{attribute 'linkalways'} 
{attribute 'no_explicit_call' := 'This FB is a CLASS and must be accessed using methods or properties'}
{attribute 'enable_dynamic_creation'}
FUNCTION_BLOCK FINAL XOR_BYTE EXTENDS Node
VAR
	in1 : _BYTE(0);
	in2 : _BYTE(0);
	out : _BYTE(0);
END_VAR

METHOD PUBLIC Clone : I_Node
VAR
	pNode : POINTER TO XOR_BYTE;
END_VAR
pNode := __NEW(XOR_BYTE);
Clone := pNode^;
END_METHOD

METHOD FB_init : BOOL
VAR_INPUT
	bInitRetains : BOOL; // if TRUE, the retain variables are initialized (warm start / cold start)
	bInCopyCode : BOOL;  // if TRUE, the instance afterwards gets moved into the copy code (online change)
END_VAR
AddInput('in1',THIS^.in1);
AddInput('in2',THIS^.in2);
AddOutput('out', THIS^.out);
END_METHOD

METHOD PROTECTED OnExecute
VAR
END_VAR
out.Value := in1.Value XOR in2.Value;
END_METHOD

END_FUNCTION_BLOCK

(* stored: Version 1.1.0.1, ProductVersion 3.1.4024.15
   POU XOR_BYTE: Id {45796d8b-2e7a-4d20-ac19-69967073d21b}, SpecialFunc None
   Folder Constructor: Id {856a0c9a-8278-4c99-951a-6edf8ae1711c}
   Method Clone: Id {8dffed33-be2a-44f9-b4ef-6653f842867c}
   Method FB_init: Id {e8e1b5d8-2dfe-4b9d-9462-6a229cb8342c}
   Method OnExecute: Id {247918e3-e920-43ab-9d2c-c9bd769eced0} *)
